PROGRAM MAIN
VAR
	ObjRunnerTestSuite : RunnerTestSuite;
END_VAR

ObjRunnerTestSuite();

END_PROGRAM

(* stored: Version 1.1.0.1
   POU MAIN: Id {1aff5ec7-e3ce-4154-9d2a-76e92eab0183}, SpecialFunc None *)
